// DUTs/ST_vertical_levitation_control_X_T
(* Generated from type 'vertical_levitation_control_X_T' *)
{attribute 'TcIecLibraryType'}
TYPE ST_vertical_levitation_control_X_T : 
	STRUCT
		(* Generated from item 'Integrator1_CSTATE' *)
		aIntegrator1_CSTATE : T_matrix4xdouble;
		(* Generated from item 'Integrator_CSTATE' *)
		fIntegrator_CSTATE : LREAL;
		(* Generated from item 'Filter_CSTATE' *)
		fFilter_CSTATE : LREAL;
		(* Generated from item 'error_integrator_CSTATE' *)
		ferror_integrator_CSTATE : LREAL;
		(* Generated from item 'time_integrator_CSTATE' *)
		ftime_integrator_CSTATE : LREAL;
		(* Generated from item 'Integrator_CSTATE_p' *)
		fIntegrator_CSTATE_p : LREAL;
		(* Generated from item 'Filtertot_CSTATE' *)
		fFiltertot_CSTATE : LREAL;
		(* Generated from item 'Integrator_CSTATE_k' *)
		fIntegrator_CSTATE_k : LREAL;
		(* Generated from item 'Filterroll_CSTATE' *)
		fFilterroll_CSTATE : LREAL;
		(* Generated from item 'Integrator_CSTATE_pl' *)
		fIntegrator_CSTATE_pl : LREAL;
		(* Generated from item 'Filterpit_CSTATE' *)
		fFilterpit_CSTATE : LREAL;
		(* Generated from item 'Integrator_CSTATE_c' *)
		fIntegrator_CSTATE_c : LREAL;
		(* Generated from item 'Filter_CSTATE_j' *)
		fFilter_CSTATE_j : LREAL;
		(* Generated from item 'Integrator_CSTATE_pq' *)
		fIntegrator_CSTATE_pq : LREAL;
		(* Generated from item 'Filter_CSTATE_b' *)
		fFilter_CSTATE_b : LREAL;
		(* Generated from item 'Integrator2_CSTATE' *)
		aIntegrator2_CSTATE : T_matrix4xdouble;
	END_STRUCT
END_TYPE

// DUTs/ST_vertical_levitation_control_DW_T
(* Generated from type 'vertical_levitation_control_DW_T' *)
{attribute 'TcIecLibraryType'}
TYPE ST_vertical_levitation_control_DW_T : 
	STRUCT
		(* Generated from item 'UnitDelay_DSTATE' *)
		aUnitDelay_DSTATE : T_matrix4xdouble;
		(* Generated from item 'Delay_DSTATE' *)
		aDelay_DSTATE : T_matrix3xdouble;
		(* Generated from item 'UnitDelay1_DSTATE' *)
		fUnitDelay1_DSTATE : LREAL;
		(* Generated from item 'UnitDelay1_DSTATE_a' *)
		fUnitDelay1_DSTATE_a : LREAL;
		(* Generated from item 'UD_DSTATE' *)
		fUD_DSTATE : LREAL;
		(* Generated from item 'UnitDelay1_DSTATE_j' *)
		fUnitDelay1_DSTATE_j : LREAL;
		(* Generated from item 'UnitDelay1_DSTATE_e' *)
		fUnitDelay1_DSTATE_e : LREAL;
		(* Generated from item 'UnitDelay1_DSTATE_ev' *)
		fUnitDelay1_DSTATE_ev : LREAL;
		(* Generated from item 'UnitDelay1_DSTATE_c' *)
		fUnitDelay1_DSTATE_c : LREAL;
		(* Generated from item 'UnitDelay1_DSTATE_d' *)
		fUnitDelay1_DSTATE_d : LREAL;
		(* Generated from item 'UnitDelay2_DSTATE' *)
		fUnitDelay2_DSTATE : LREAL;
		(* Generated from item 'UnitDelay2_DSTATE_l' *)
		fUnitDelay2_DSTATE_l : LREAL;
		(* Generated from item 'UnitDelay2_DSTATE_lt' *)
		fUnitDelay2_DSTATE_lt : LREAL;
		(* Generated from item 'UnitDelay2_DSTATE_j' *)
		fUnitDelay2_DSTATE_j : LREAL;
		(* Generated from item 'Delay1_DSTATE' *)
		fDelay1_DSTATE : REAL;
		(* Generated from item 'Memory_PreviousInput' *)
		bMemory_PreviousInput : BOOL;
		(* Generated from item 'Memory_PreviousInput_l' *)
		bMemory_PreviousInput_l : BOOL;
		(* Generated from item 'Memory_PreviousInput_a' *)
		bMemory_PreviousInput_a : BOOL;
		 {attribute 'hide'}
		_reserved1 : USINT;
	END_STRUCT
END_TYPE

// DUTs/ST_GetSet_OTCID
{attribute 'TcIecLibraryType'}
{attribute 'hide'}
TYPE ST_GetSet_OTCID : 
	STRUCT
		{attribute 'GUID' := '18071995-0000-0000-0000-000000000018'}
		{attribute 'GlobalType'}
		pInst : PVOID;
		{attribute 'GUID' := '18071995-0000-0000-0000-00000000000F'}
		{attribute 'GlobalType'}
		nParam : OTCID;
		 {attribute 'hide'}
		_reserved1 : UINT_0_32;
	END_STRUCT
END_TYPE

// DUTs/ST_GetSet_UDINT
{attribute 'TcIecLibraryType'}
{attribute 'hide'}
TYPE ST_GetSet_UDINT : 
	STRUCT
		{attribute 'GUID' := '18071995-0000-0000-0000-000000000018'}
		{attribute 'GlobalType'}
		pInst : PVOID;
		nParam : UDINT;
		 {attribute 'hide'}
		_reserved1 : UINT_0_32;
	END_STRUCT
END_TYPE

// DUTs/ST_GetSet_UINT
{attribute 'TcIecLibraryType'}
{attribute 'hide'}
TYPE ST_GetSet_UINT : 
	STRUCT
		{attribute 'GUID' := '18071995-0000-0000-0000-000000000018'}
		{attribute 'GlobalType'}
		pInst : PVOID;
		nParam : UINT;
		 {attribute 'hide'}
		_reserved1 : UINT_16_48;
	END_STRUCT
END_TYPE

// DUTs/ST_GetSet_TcTraceLevel
{attribute 'TcIecLibraryType'}
{attribute 'hide'}
TYPE ST_GetSet_TcTraceLevel : 
	STRUCT
		{attribute 'GUID' := '18071995-0000-0000-0000-000000000018'}
		{attribute 'GlobalType'}
		pInst : PVOID;
		{attribute 'GUID' := '8007AE3B-86BB-40F2-B385-EF87FCC239A4'}
		{attribute 'GlobalType'}
		eParam : TcTraceLevel;
		 {attribute 'hide'}
		_reserved1 : UINT_0_32;
	END_STRUCT
END_TYPE

// DUTs/ST_GetSet_E_ModuleCaller
{attribute 'TcIecLibraryType'}
{attribute 'hide'}
TYPE ST_GetSet_E_ModuleCaller : 
	STRUCT
		{attribute 'GUID' := '18071995-0000-0000-0000-000000000018'}
		{attribute 'GlobalType'}
		pInst : PVOID;
		eParam : E_ModuleCaller;
		 {attribute 'hide'}
		_reserved1 : UINT_0_32;
	END_STRUCT
END_TYPE

// DUTs/ST_GetSet_E_CallerVerification
{attribute 'TcIecLibraryType'}
{attribute 'hide'}
TYPE ST_GetSet_E_CallerVerification : 
	STRUCT
		{attribute 'GUID' := '18071995-0000-0000-0000-000000000018'}
		{attribute 'GlobalType'}
		pInst : PVOID;
		eParam : E_CallerVerification;
		 {attribute 'hide'}
		_reserved1 : UINT_0_32;
	END_STRUCT
END_TYPE

// DUTs/ST_GetSet_E_StepSizeAdaptation
{attribute 'TcIecLibraryType'}
{attribute 'hide'}
TYPE ST_GetSet_E_StepSizeAdaptation : 
	STRUCT
		{attribute 'GUID' := '18071995-0000-0000-0000-000000000018'}
		{attribute 'GlobalType'}
		pInst : PVOID;
		eParam : E_StepSizeAdaptation;
		 {attribute 'hide'}
		_reserved1 : UINT_0_32;
	END_STRUCT
END_TYPE

// DUTs/ST_GetSet_E_ExecutionSequence1
{attribute 'TcIecLibraryType'}
{attribute 'hide'}
TYPE ST_GetSet_E_ExecutionSequence1 : 
	STRUCT
		{attribute 'GUID' := '18071995-0000-0000-0000-000000000018'}
		{attribute 'GlobalType'}
		pInst : PVOID;
		eParam : E_ExecutionSequence1;
		 {attribute 'hide'}
		_reserved1 : UINT_0_32;
	END_STRUCT
END_TYPE

// DUTs/ST_GetSet_E_FpExcptCtrlSet
{attribute 'TcIecLibraryType'}
{attribute 'hide'}
TYPE ST_GetSet_E_FpExcptCtrlSet : 
	STRUCT
		{attribute 'GUID' := '18071995-0000-0000-0000-000000000018'}
		{attribute 'GlobalType'}
		pInst : PVOID;
		eParam : E_FpExcptCtrlSet;
		 {attribute 'hide'}
		_reserved1 : UINT_24_56;
	END_STRUCT
END_TYPE

// DUTs/ST_ModuleBuildInfo
(* Generated from type 'TcMgSdk.ModuleBuildInfo' *)
{attribute 'TcIecLibraryType'}
TYPE ST_ModuleBuildInfo : 
	STRUCT
		(* Generated from item 'TcBuild' *)
		nTcBuild : UDINT;
		(* Generated from item 'TcRevision' *)
		nTcRevision : UDINT;
		(* Generated from item 'Debug' *)
		bDebug : BOOL;
		 {attribute 'hide'}
		_reserved1 : ARRAY [1..3] OF USINT;
	END_STRUCT
END_TYPE

// DUTs/ST_GetSet_ST_ModuleBuildInfo
{attribute 'TcIecLibraryType'}
{attribute 'hide'}
TYPE ST_GetSet_ST_ModuleBuildInfo : 
	STRUCT
		{attribute 'GUID' := '18071995-0000-0000-0000-000000000018'}
		{attribute 'GlobalType'}
		pInst : PVOID;
		stParam : ST_ModuleBuildInfo;
		 {attribute 'hide'}
		_reserved1 : UINT_0_32;
	END_STRUCT
END_TYPE

// DUTs/ST_LibraryInfo
(* Generated from type 'TcMgSdk.LibraryInfo' *)
{attribute 'TcIecLibraryType'}
TYPE ST_LibraryInfo : 
	STRUCT
		(* Generated from item 'FileVersion' *)
		nFileVersion : ARRAY [0..3] OF UDINT;
		(* Generated from item 'ProductVersion' *)
		nProductVersion : ARRAY [0..3] OF UDINT;
		(* Generated from item 'VendorName' *)
		{attribute 'GUID' := '18071995-0000-0000-0000-00010000007F'}
		{attribute 'GlobalType'}
		sVendorName : STRING(127);
		(* Generated from item 'LibraryName' *)
		{attribute 'GUID' := '18071995-0000-0000-0000-00010000007F'}
		{attribute 'GlobalType'}
		sLibraryName : STRING(127);
		(* Generated from item 'LibraryVersion' *)
		nLibraryVersion : ARRAY [0..3] OF UDINT;
		(* Generated from item 'LibraryId' *)
		{attribute 'GUID' := '18071995-0000-0000-0000-00010000007F'}
		{attribute 'GlobalType'}
		sLibraryId : STRING(127);
		(* Generated from item 'LibraryGUID' *)
		{attribute 'GUID' := '18071995-0000-0000-0000-000000000024'}
		{attribute 'GlobalType'}
		nLibraryGUID : CLSID;
		(* Generated from item 'TcSdkVersion' *)
		nTcSdkVersion : ARRAY [0..3] OF UDINT;
		(* Generated from item 'Compiler' *)
		{attribute 'GUID' := '18071995-0000-0000-0000-00010000007F'}
		{attribute 'GlobalType'}
		sCompiler : STRING(127);
		(* Generated from item 'Debug' *)
		bDebug : BOOL;
		 {attribute 'hide'}
		_reserved1 : ARRAY [1..7] OF USINT;
	END_STRUCT
END_TYPE

// DUTs/ST_GetSet_ST_LibraryInfo
{attribute 'TcIecLibraryType'}
{attribute 'hide'}
TYPE ST_GetSet_ST_LibraryInfo : 
	STRUCT
		{attribute 'GUID' := '18071995-0000-0000-0000-000000000018'}
		{attribute 'GlobalType'}
		pInst : PVOID;
		stParam : ST_LibraryInfo;
	END_STRUCT
END_TYPE

// DUTs/ST_ModuleInfo
(* Generated from type 'TcMgSdk.ModuleInfo' *)
{attribute 'TcIecLibraryType'}
TYPE ST_ModuleInfo : 
	STRUCT
		(* Generated from item 'ClassName' *)
		{attribute 'GUID' := '18071995-0000-0000-0000-00010000007F'}
		{attribute 'GlobalType'}
		sClassName : STRING(127);
		(* Generated from item 'CommonClassId' *)
		{attribute 'GUID' := '18071995-0000-0000-0000-000000000024'}
		{attribute 'GlobalType'}
		nCommonClassId : CLSID;
		(* Generated from item 'VersionClassId' *)
		{attribute 'GUID' := '18071995-0000-0000-0000-000000000024'}
		{attribute 'GlobalType'}
		nVersionClassId : CLSID;
	END_STRUCT
END_TYPE

// DUTs/ST_GetSet_ST_ModuleInfo
{attribute 'TcIecLibraryType'}
{attribute 'hide'}
TYPE ST_GetSet_ST_ModuleInfo : 
	STRUCT
		{attribute 'GUID' := '18071995-0000-0000-0000-000000000018'}
		{attribute 'GlobalType'}
		pInst : PVOID;
		stParam : ST_ModuleInfo;
	END_STRUCT
END_TYPE

// DUTs/ST_GetSet_ST_TcMatSim_ModuleGeneratorInfo
{attribute 'TcIecLibraryType'}
{attribute 'hide'}
TYPE ST_GetSet_ST_TcMatSim_ModuleGeneratorInfo : 
	STRUCT
		{attribute 'GUID' := '18071995-0000-0000-0000-000000000018'}
		{attribute 'GlobalType'}
		pInst : PVOID;
		stParam : ST_TcMatSim_ModuleGeneratorInfo;
	END_STRUCT
END_TYPE

// DUTs/ST_GetSet_ST_TcMatSim_SimulinkModelInfo
{attribute 'TcIecLibraryType'}
{attribute 'hide'}
TYPE ST_GetSet_ST_TcMatSim_SimulinkModelInfo : 
	STRUCT
		{attribute 'GUID' := '18071995-0000-0000-0000-000000000018'}
		{attribute 'GlobalType'}
		pInst : PVOID;
		stParam : ST_TcMatSim_SimulinkModelInfo;
	END_STRUCT
END_TYPE

// DUTs/ST_GetSet_E_ParameterSharingType
{attribute 'TcIecLibraryType'}
{attribute 'hide'}
TYPE ST_GetSet_E_ParameterSharingType : 
	STRUCT
		{attribute 'GUID' := '18071995-0000-0000-0000-000000000018'}
		{attribute 'GlobalType'}
		pInst : PVOID;
		eParam : E_ParameterSharingType;
		 {attribute 'hide'}
		_reserved1 : UINT_0_32;
	END_STRUCT
END_TYPE

// DUTs/ST_GetSet_ST_P_vertical_levitation_control_T
{attribute 'TcIecLibraryType'}
{attribute 'hide'}
TYPE ST_GetSet_ST_P_vertical_levitation_control_T : 
	STRUCT
		{attribute 'GUID' := '18071995-0000-0000-0000-000000000018'}
		{attribute 'GlobalType'}
		pInst : PVOID;
		stParam : ST_P_vertical_levitation_control_T;
	END_STRUCT
END_TYPE

// DUTs/ST_GetSet_LREAL
{attribute 'TcIecLibraryType'}
{attribute 'hide'}
TYPE ST_GetSet_LREAL : 
	STRUCT
		{attribute 'GUID' := '18071995-0000-0000-0000-000000000018'}
		{attribute 'GlobalType'}
		pInst : PVOID;
		fParam : LREAL;
	END_STRUCT
END_TYPE

// Version/Global_Version
{attribute 'TcGenerated'}
// This function has been automatically generated from the project information.
VAR_GLOBAL CONSTANT
	{attribute 'const_non_replaced'}
	{attribute 'linkalways'}
	stLibVersion_vertical_levitation_control : ST_LibVersion := (iMajor := 0, iMinor := 0, iBuild := 0, iRevision := 27, nFlags := 0, sVersion := '0.0.0.27');
	{attribute 'const_non_replaced'}
	{attribute 'linkalways'}
	sLibraryId_vertical_levitation_control : String := 'TE140x Module Vendor|vertical_levitation_control|0.0.0.27';
END_VAR

// POUs/FB_vertical_levitation_control

{attribute 'c++_compatible'}
{attribute 'external_name' := 'FB_vertical_levitation_control_GUID_57ABDA4F_9E3A_C8D3_BBCC_2358706B3C72'}
{attribute 'TcIecLibraryType'}
{attribute 'reflection'}
FUNCTION_BLOCK FB_vertical_levitation_control
VAR
	{attribute 'hide'}
	{attribute 'no_copy'}
	{attribute 'GUID' := '18071995-0000-0000-0000-000000000018'}
	{attribute 'GlobalType'}
	m_pData : PVOID;
	{attribute 'TcInitSymbol'}
	{attribute 'GUID' := '8007AE3B-86BB-40F2-B385-EF87FCC239A4'}
	{attribute 'GlobalType'}
	eTraceLevelMax : TcTraceLevel := TcTraceLevel.tlInfo;
	 {attribute 'hide'}
	_reserved1 : UDINT;
	{attribute 'hide'}
	{attribute 'instance-path'}
	{attribute 'noinit'}
	{attribute 'GUID' := '18071995-0000-0000-0000-0001000000FF'}
	{attribute 'GlobalType'}
	sInstancePath : STRING(255);
	{attribute 'hide'}
	{attribute 'noinit'}
	{attribute 'GUID' := '18071995-0000-0000-0000-000000000019'}
	{attribute 'GlobalType'}
	m_HResultLog : HRESULT;
	{attribute 'hide'}
	{attribute 'noinit'}
	{attribute 'GUID' := '18071995-0000-0000-0000-000000000019'}
	{attribute 'GlobalType'}
	m_HResult : HRESULT;
	 {attribute 'hide'}
	_reserved2 : ARRAY [1..184] OF USINT;
	{attribute 'hide'}
	{attribute 'no_copy'}
	m_ExtModeData : ULINT;
END_VAR
VAR_INPUT
	(* Generated from item 'z_avg' *)
	fz_avg : LREAL;
	(* Generated from item 'roll_measured' *)
	froll_measured : LREAL;
	(* Generated from item 'pitch_measured' *)
	fpitch_measured : LREAL;
	(* Generated from item 'ems_roll' *)
	fems_roll : LREAL;
	(* Generated from item 'F_imu' *)
	aF_imu : T_matrix3xdouble;
	(* Generated from item 'gyro_imu' *)
	agyro_imu : T_matrix3xdouble;
	(* Generated from item 'motor_Fy_l' *)
	fmotor_Fy_l : LREAL;
	(* Generated from item 'motor_Fy_r' *)
	fmotor_Fy_r : LREAL;
END_VAR
VAR_OUTPUT
	(* Generated from item 'I_VFL' *)
	aI_VFL : T_matrix2xdouble;
	(* Generated from item 'I_VFR' *)
	aI_VFR : T_matrix2xdouble;
	(* Generated from item 'I_VBL' *)
	aI_VBL : T_matrix2xdouble;
	(* Generated from item 'I_VBR' *)
	aI_VBR : T_matrix2xdouble;
	(* Generated from item 'F_hems' *)
	aF_hems : T_matrix4xdouble;
	(* Generated from item 'F_requested' *)
	aF_requested : T_matrix3xdouble;
	(* Generated from item 'integral_terms' *)
	aintegral_terms : T_matrix3xdouble;
	(* Generated from item 'sat_failed' *)
	fsat_failed : LREAL;
	(* Generated from item 'net_post_sat' *)
	anet_post_sat : T_matrix3xdouble;
	(* Generated from item 'z_target_adjusted' *)
	fz_target_adjusted : LREAL;
	(* Generated from item 'Max_allowed_current' *)
	aMax_allowed_current : T_matrix4xdouble;
	(* Generated from item 'Min_allowed_current' *)
	aMin_allowed_current : T_matrix4xdouble;
END_VAR
VAR
	{attribute 'no_copy'}
	Pvertical_levitation_control_M : POINTER TO ST_RT_MODEL_vertical_levitation_control_T;
END_VAR

{attribute 'TcTypeSystem'}

METHOD FB_exit : BOOL
VAR_INPUT
	bInCopyCode : BOOL;
END_VAR
END_METHOD

{attribute 'TcTypeSystem'}

METHOD FB_init : BOOL
VAR_INPUT
	bInitRetains : BOOL;
	bInCopyCode : BOOL;
END_VAR
END_METHOD

{attribute 'TcTypeSystem'}

{attribute 'monitoring' := 'call'}
	PROPERTY nHResult : HRESULT
GET
END_GET
END_PROPERTY

{attribute 'TcTypeSystem'}

{attribute 'monitoring' := 'call'}
	PROPERTY eInitExceptionHandling : E_FpExcptCtrlSetEx
GET
END_GET
SET
END_SET
END_PROPERTY

{attribute 'TcTypeSystem'}

{attribute 'monitoring' := 'call'}
	PROPERTY eUpdateExceptionHandling : E_FpExcptCtrlSetEx
GET
END_GET
SET
END_SET
END_PROPERTY

{attribute 'TcTypeSystem'}

{attribute 'monitoring' := 'call'}
	PROPERTY nExceptionCnt : ULINT
GET
END_GET
END_PROPERTY

{attribute 'TcTypeSystem'}

{attribute 'monitoring' := 'variable'}
	PROPERTY stActiveException : ST_ExceptionInfo
GET
END_GET
END_PROPERTY

{attribute 'TcTypeSystem'}

{attribute 'monitoring' := 'call'}
	PROPERTY bInitialized : BOOL
GET
END_GET
END_PROPERTY

{attribute 'TcTypeSystem'}

{attribute 'monitoring' := 'call'}
	PROPERTY bExecute : BOOL
GET
END_GET
SET
END_SET
END_PROPERTY

END_FUNCTION_BLOCK

// POUs/TcCOM Wrapper/FB_vertical_levitation_control_TcCOM_InitStruct

{attribute 'c++_compatible'}
{attribute 'external_name' := 'FB_vertical_levitation_control_TcCOM_InitStruct_GUID_A1358BCC_0A9B_2D17_1AF2_27948DBD901E'}
{attribute 'TcIecLibraryType'}
{attribute 'call_after_init'}
{attribute 'reflection'}
FUNCTION_BLOCK FB_vertical_levitation_control_TcCOM_InitStruct
VAR
	{attribute 'hide'}
	{attribute 'no_copy'}
	{attribute 'GUID' := '18071995-0000-0000-0000-000000000018'}
	{attribute 'GlobalType'}
	m_pData : PVOID;
	{attribute 'TcInitSymbol'}
	{attribute 'GUID' := '8007AE3B-86BB-40F2-B385-EF87FCC239A4'}
	{attribute 'GlobalType'}
	eTraceLevelMaxFB : TcTraceLevel := TcTraceLevel.tlInfo;
	 {attribute 'hide'}
	_reserved1 : UDINT;
	{attribute 'hide'}
	{attribute 'instance-path'}
	{attribute 'noinit'}
	{attribute 'GUID' := '18071995-0000-0000-0000-0001000000FF'}
	{attribute 'GlobalType'}
	sInstancePath : STRING(255);
	{attribute 'hide'}
	{attribute 'noinit'}
	{attribute 'GUID' := '18071995-0000-0000-0000-000000000019'}
	{attribute 'GlobalType'}
	m_HResultLog : HRESULT;
	{attribute 'hide'}
	{attribute 'noinit'}
	{attribute 'GUID' := '18071995-0000-0000-0000-000000000019'}
	{attribute 'GlobalType'}
	m_HResult : HRESULT;
	 {attribute 'hide'}
	_reserved2 : UINT_0_32;
	 {attribute 'hide'}
	_reserved3 : ARRAY [1..12] OF UINT_8_16;
	 {attribute 'hide'}
	_reserved4 : ARRAY [1..12] OF USINT;
END_VAR
VAR_INPUT
	stvertical_levitation_control_U : ST_vertical_levitation_control_U_T;
END_VAR
VAR_OUTPUT
	stvertical_levitation_control_Y : ST_vertical_levitation_control_Y_T;
END_VAR
VAR
	{attribute 'hide'}
	{attribute 'GUID' := '7C96C7D1-E238-BB86-5119-B8C749E25768'}
	_ipvertical_levitation_control : POINTER TO ITcvertical_levitation_control;
	stInit : ST_FB_vertical_levitation_control_TcCOM_InitStruct;
END_VAR

{attribute 'TcTypeSystem'}

METHOD FB_init : BOOL
VAR_INPUT
	bInitRetains : BOOL;
	bInCopyCode : BOOL;
	{attribute 'GUID' := 'EC8BF77E-C48E-D37A-9903-A8E87F5E2714'}
	stInit : REFERENCE TO ST_FB_vertical_levitation_control_TcCOM_InitStruct;
END_VAR
END_METHOD

{attribute 'TcTypeSystem'}

{attribute 'call_after_init'}
METHOD FB_afterinit : BOOL
END_METHOD

{attribute 'TcTypeSystem'}

METHOD Reinit : BOOL
VAR_INPUT
	{attribute 'GUID' := 'EC8BF77E-C48E-D37A-9903-A8E87F5E2714'}
	stReInit : ST_FB_vertical_levitation_control_TcCOM_InitStruct;
END_VAR
END_METHOD

{attribute 'TcTypeSystem'}

METHOD FB_exit : BOOL
VAR_INPUT
	bInCopyCode : BOOL;
END_VAR
END_METHOD

{attribute 'TcTypeSystem'}

	PROPERTY eObjectState : TCOM_STATE
GET
END_GET
SET
END_SET
END_PROPERTY

{attribute 'TcTypeSystem'}

{attribute 'monitoring' := 'call'}
	PROPERTY nHResult : HRESULT
GET
END_GET
END_PROPERTY

{attribute 'TcTypeSystem'}

	PROPERTY ipTcComObject : ITComObject
GET
END_GET
END_PROPERTY

{attribute 'TcTypeSystem'}

	PROPERTY ipADI : ITcADI
GET
END_GET
END_PROPERTY

{attribute 'TcTypeSystem'}

{attribute 'monitoring' := 'call'}
	PROPERTY nTaskOid : OTCID
GET
END_GET
SET
END_SET
END_PROPERTY

{attribute 'TcTypeSystem'}

{attribute 'monitoring' := 'call'}
	PROPERTY nTaskPriority : UDINT
GET
END_GET
END_PROPERTY

{attribute 'TcTypeSystem'}

{attribute 'monitoring' := 'call'}
	PROPERTY nTaskCycleTimeNs : UDINT
GET
END_GET
END_PROPERTY

{attribute 'TcTypeSystem'}

{attribute 'monitoring' := 'call'}
	PROPERTY nTaskPort : UINT
GET
END_GET
END_PROPERTY

{attribute 'TcTypeSystem'}

{attribute 'monitoring' := 'call'}
	PROPERTY nTaskSortOrder : UDINT
GET
END_GET
SET
END_SET
END_PROPERTY

{attribute 'TcTypeSystem'}

{attribute 'monitoring' := 'call'}
	PROPERTY eTraceLevelMax : TcTraceLevel
GET
END_GET
SET
END_SET
END_PROPERTY

{attribute 'TcTypeSystem'}

{attribute 'monitoring' := 'call'}
	PROPERTY eModuleCaller : E_ModuleCaller
GET
END_GET
SET
END_SET
END_PROPERTY

{attribute 'TcTypeSystem'}

{attribute 'monitoring' := 'call'}
	PROPERTY eCallerVerification : E_CallerVerification
GET
END_GET
SET
END_SET
END_PROPERTY

{attribute 'TcTypeSystem'}

{attribute 'monitoring' := 'call'}
	PROPERTY eStepSizeAdaptation : E_StepSizeAdaptation
GET
END_GET
SET
END_SET
END_PROPERTY

{attribute 'TcTypeSystem'}

{attribute 'monitoring' := 'call'}
	PROPERTY eExecutionSequence : E_ExecutionSequence1
GET
END_GET
SET
END_SET
END_PROPERTY

{attribute 'TcTypeSystem'}

{attribute 'monitoring' := 'call'}
	PROPERTY bExecute : BOOL
GET
END_GET
SET
END_SET
END_PROPERTY

{attribute 'TcTypeSystem'}

{attribute 'monitoring' := 'call'}
	PROPERTY eAccessLockState : TCOM_STATE
GET
END_GET
SET
END_SET
END_PROPERTY

{attribute 'TcTypeSystem'}

{attribute 'monitoring' := 'call'}
	PROPERTY eInitExceptionHandling : E_FpExcptCtrlSet
GET
END_GET
SET
END_SET
END_PROPERTY

{attribute 'TcTypeSystem'}

{attribute 'monitoring' := 'call'}
	PROPERTY eUpdateExceptionHandling : E_FpExcptCtrlSetEx
GET
END_GET
SET
END_SET
END_PROPERTY

{attribute 'TcTypeSystem'}

{attribute 'monitoring' := 'variable'}
	PROPERTY stModuleBuildInfo : ST_ModuleBuildInfo
GET
END_GET
END_PROPERTY

{attribute 'TcTypeSystem'}

{attribute 'monitoring' := 'call'}
	PROPERTY bInitialized : BOOL
GET
END_GET
END_PROPERTY

{attribute 'TcTypeSystem'}

{attribute 'monitoring' := 'call'}
	PROPERTY nSkippedExecutionCount : UDINT
GET
END_GET
END_PROPERTY

{attribute 'TcTypeSystem'}

{attribute 'monitoring' := 'variable'}
	PROPERTY stLibraryInfo : ST_LibraryInfo
GET
END_GET
END_PROPERTY

{attribute 'TcTypeSystem'}

{attribute 'monitoring' := 'variable'}
	PROPERTY stModuleInfo : ST_ModuleInfo
GET
END_GET
END_PROPERTY

{attribute 'TcTypeSystem'}

{attribute 'monitoring' := 'variable'}
	PROPERTY stModuleGeneratorInfo : ST_TcMatSim_ModuleGeneratorInfo
GET
END_GET
SET
END_SET
END_PROPERTY

{attribute 'TcTypeSystem'}

{attribute 'monitoring' := 'variable'}
	PROPERTY stSimulinkModelInfo : ST_TcMatSim_SimulinkModelInfo
GET
END_GET
SET
END_SET
END_PROPERTY

{attribute 'TcTypeSystem'}

{attribute 'monitoring' := 'call'}
	PROPERTY evertical_levitation_control_P_Sharing : E_ParameterSharingType
GET
END_GET
SET
END_SET
END_PROPERTY

{attribute 'TcTypeSystem'}

{attribute 'monitoring' := 'call'}
	PROPERTY nvertical_levitation_control_P_Definer : OTCID
GET
END_GET
END_PROPERTY

{attribute 'TcTypeSystem'}

{attribute 'monitoring' := 'variable'}
	PROPERTY stvertical_levitation_control_P : ST_P_vertical_levitation_control_T
GET
END_GET
SET
END_SET
END_PROPERTY

{attribute 'TcTypeSystem'}

{attribute 'monitoring' := 'call'}
	PROPERTY fSimulationTime : LREAL
GET
END_GET
END_PROPERTY

{attribute 'TcTypeSystem'}

{attribute 'monitoring' := 'call'}
	PROPERTY nCycleCount : ULINT
GET
END_GET
END_PROPERTY

{attribute 'TcTypeSystem'}

{attribute 'monitoring' := 'call'}
	PROPERTY nExceptionCount : ULINT
GET
END_GET
END_PROPERTY

{attribute 'TcTypeSystem'}

{attribute 'monitoring' := 'variable'}
	PROPERTY stExceptionInfo : ST_ExceptionInfo
GET
END_GET
END_PROPERTY

END_FUNCTION_BLOCK
